{attribute 'linkalways'} 
{attribute 'no_explicit_call' := 'This FB is a CLASS and must be accessed using methods or properties'}
{attribute 'enable_dynamic_creation'}
FUNCTION_BLOCK _FLOAT EXTENDS AliasDatatypeBase
VAR
	localData : FLOAT;
	activeData : REFERENCE TO FLOAT REF= localData;
	aliasBaseDatatype : _LREAL(localData);
END_VAR

PROPERTY PUBLIC Address : PVOID
GET
Address := ADR(activeData);
END_GET
END_PROPERTY

METHOD PUBLIC ClearReference
VAR_INPUT
END_VAR
activeData REF= localData;
SetBaseDatatypeReference();
END_METHOD

METHOD PUBLIC Clone : I_Datatype
VAR
    pClone : POINTER TO _FLOAT;
END_VAR
pClone := __NEW(_FLOAT(InitialValue := Value));
Clone := pClone^;
END_METHOD

METHOD FB_init : BOOL
VAR_INPUT
	bInitRetains : BOOL; // if TRUE, the retain variables are initialized (warm start / cold start)
	bInCopyCode : BOOL;  // if TRUE, the instance afterwards gets moved into the copy code (online change)
	InitialValue : FLOAT;
END_VAR
localData := InitialValue;
SetBaseDatatypeReference();
AddBaseDatatype(aliasBaseDatatype);
END_METHOD

PROPERTY PUBLIC Identifier : T_MAXSTRING
GET
Identifier := 'FLOAT';
END_GET
END_PROPERTY

METHOD PUBLIC MakeReferenceTo
VAR_INPUT
	ReferenceTarget : REFERENCE TO FLOAT;
END_VAR
activeData REF= ReferenceTarget;
SetBaseDatatypeReference();
END_METHOD

METHOD PROTECTED SetBaseDatatypeReference
VAR_INPUT
END_VAR
aliasBaseDatatype.MakeReferenceTo(activeData);
END_METHOD

PROPERTY PUBLIC Size : UDINT
GET
Size := SIZEOF(activeData);
END_GET
END_PROPERTY

METHOD TryMakeReferenceTo : BOOL
VAR_INPUT
	Target : I_Datatype;
END_VAR
VAR
	targetAsAlias : I_AliasDatatype;
	pTargetData : POINTER TO FLOAT;
END_VAR
IF NOT Target.TryResolveAsAliasDatatype(targetAsAlias) THEN
	RETURN;
END_IF

IF targetAsAlias.Identifier <> Identifier THEN
	RETURN;
END_IF

pTargetData := Target.Address;
activeData REF= pTargetData^;
SetBaseDatatypeReference();
TryMakeReferenceTo := TRUE;
END_METHOD

PROPERTY PUBLIC Value : REFERENCE TO FLOAT
GET
Value REF= activeData;
END_GET
END_PROPERTY

END_FUNCTION_BLOCK

(* stored: Version 1.1.0.1, ProductVersion 3.1.4024.12
   POU _FLOAT: Id {15cd4300-120a-4ff8-af41-d93d4c835e03}, SpecialFunc None
   Folder Constructor: Id {aba9d7a7-325d-454a-b66c-99639ab7b72a}
   Folder Protected: Id {6b3ea4e6-e4e4-4283-bd4d-fbadc268fa39}
   Property Address: Id {d7fa9739-8b96-4eba-8472-4801c5b26fc1}
   Get Get: Id {ec4d86a3-df2e-4574-b2c6-df2b04cd7350}
   Method ClearReference: Id {543e86c3-7825-46b0-b9dd-59c27d480a9b}
   Method Clone: Id {42140205-0604-4c67-ae77-9b6080da6cd2}
   Method FB_init: Id {7cc8a50f-6146-42fd-b3ec-91b31ba4737e}
   Property Identifier: Id {fcb59706-6847-41f2-90d1-3c5bc8e48020}
   Get Get: Id {1d745473-d8d5-4076-b07d-bdefe74adfc0}
   Method MakeReferenceTo: Id {077594aa-b343-41a1-96eb-32a30bbc52f6}
   Method SetBaseDatatypeReference: Id {b775926a-1b91-433a-80a2-0e9ff3ebf0b9}
   Property Size: Id {70b1eba6-15d1-4bfb-834e-a647c7343825}
   Get Get: Id {0d2f028d-1bc2-4847-bbd5-341edd996ea2}
   Method TryMakeReferenceTo: Id {8c2ad742-ea1a-43cb-92fb-71c1b828da6b}
   Property Value: Id {f53f00e0-1620-4ef0-8582-f59a465388d2}
   Get Get: Id {615b3c0c-2c82-4e4b-895f-0fadfbef4cb9} *)
